(* Specifies the operating mode of a controller. *)
{attribute 'qualified_only'}
{attribute 'strict'}
{attribute 'to_string'}
TYPE E_ControllerMode :
(
	// Output is computed from Setpoint and Feedback using the controller's algorithm.
	Auto 	:= 0,
	// Output tracks Setpoint directly.
	Manual	:= 1
)BYTE;
END_TYPE

(* stored: Version 1.1.0.1, ProductVersion 3.1.4024.15
   EnumerationTextList E_ControllerMode: Id {ad840b95-c69a-0b49-1cff-63e9d69bb985} *)
